TYPE "ST_SpkCylinderParCfg"
VERSION : 0.1
   STRUCT
      SchemaVersion : UInt := 1;   // Core s.3.8: first member of every ParCfg
      MoveTimeoutMs : UDInt := 2000;
   END_STRUCT;

END_TYPE
